FUNCTION_BLOCK RemoveWP
  (* Standard: 61499-2 *)
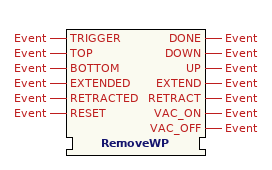
  EVENT_INPUT
    TRIGGER;
    TOP;
    BOTTOM;
    EXTENDED;
    RETRACTED;
    RESET;
  END_EVENT
  EVENT_OUTPUT
    DONE;
    DOWN;
    UP;
    EXTEND;
    RETRACT;
    VAC_ON;
    VAC_OFF;
  END_EVENT
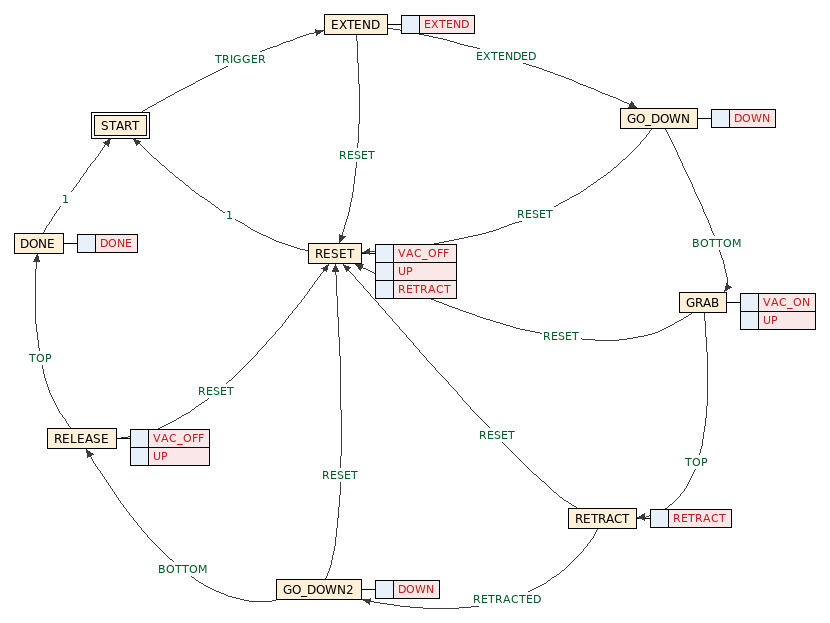
  EC_STATES
    START;
    GO_DOWN : -> DOWN;
    GRAB : -> VAC_ON, -> UP;
    EXTEND : -> EXTEND;
    GO_DOWN2 : -> DOWN;
    RELEASE : -> VAC_OFF, -> UP;
    RETRACT : -> RETRACT;
    DONE : -> DONE;
    RESET : -> VAC_OFF, -> UP, -> RETRACT;
  END_STATES
  EC_TRANSITIONS
    START TO EXTEND := TRIGGER;
    GO_DOWN TO GRAB := BOTTOM;
    GRAB TO RETRACT := TOP;
    EXTEND TO GO_DOWN := EXTENDED;
    GO_DOWN2 TO RELEASE := BOTTOM;
    RELEASE TO DONE := TOP;
    RETRACT TO GO_DOWN2 := RETRACTED;
    DONE TO START := 1;
    EXTEND TO RESET := RESET;
    GO_DOWN TO RESET := RESET;
    GRAB TO RESET := RESET;
    RETRACT TO RESET := RESET;
    GO_DOWN2 TO RESET := RESET;
    RELEASE TO RESET := RESET;
    RESET TO START := 1;
  END_TRANSITIONS
  ALGORITHM INIT IN ST:

  END_ALGORITHM
  ALGORITHM REQ IN ST:

  END_ALGORITHM
END_FUNCTION_BLOCK
